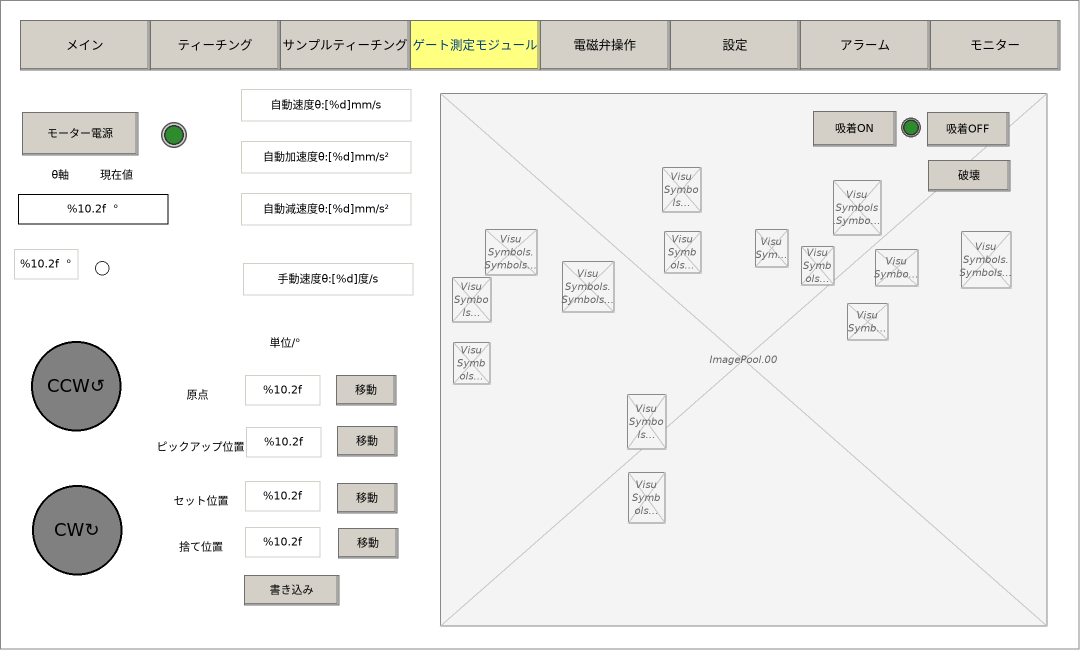
VISUALIZATION s_gm_teaching  // 1080x650
    Rectangle (0,0 1080x650)
    Label (35,160 51x30), "θ軸"
    Rectangle (18,194 150x30), "%10.2f °", text variable: gvl_axis.axisR.NcToPlc.ActPos
    Ellipse (31,341 90x90), "CCW↺", invisible if: gvl_axis.fbi_mc_powerR.Busy = FALSE
        OnMouseDown: execute { gvl_visu.flg_btn_rotaryRigt := true; }
        OnMouseUp: execute { gvl_visu.flg_btn_rotaryRigt := FALSE; }
    Ellipse (32,485 90x90), "CW↻", invisible if: gvl_axis.fbi_mc_powerR.Busy = FALSE
        OnMouseDown: execute { gvl_visu.flg_btn_rotaryLeft := TRUE; }
        OnMouseUp: execute { gvl_visu.flg_btn_rotaryLeft := FALSE; }
    Textfield (245,375 75x30), "%10.2f", text variable: gvl_visu.var_rotaryPos.origin
        OnMouseClick: write gvl_visu.var_rotaryPos.origin via VisuDialogs.Numpad
    Label (154,380 87x30), "原点"
    Textfield (246,427 75x30), "%10.2f", text variable: gvl_visu.var_rotaryPos.pickUp
        OnMouseClick: write gvl_visu.var_rotaryPos.pickUp via VisuDialogs.Numpad
    Label (159,432 83x30), "ピックアップ位置"
    Textfield (245,481 75x30), "%10.2f", text variable: gvl_visu.var_rotaryPos.set
        OnMouseClick: write gvl_visu.var_rotaryPos.set via VisuDialogs.Numpad
    Label (161,486 80x30), "セット位置"
    Lamp1 (159,120 30x30), variable: gvl_axis.fbi_mc_powerR.Busy, style: Lamp-Lamp1-Green
    Textfield (14,249 64x30), "%10.2f °", text variable: gvl_visu.var_gm_rotaryInch
        OnMouseClick: write gvl_visu.var_gm_rotaryInch via VisuDialogs.Numpad, format mm
    RadioButton (93,248 150x40), variable: gvl_visu.var_radio_rotaryJogMode
        Areas[0]: Text=インチ
        Areas[1]: Text=ジョグ
    Button (22,112 116x43), "モーター電源"
        toggle gvl_visu.flg_btn_gm_motorPower
    Button (244,575 95x30), "書き込み", colour toggle: gvl_visu.flg_btn_rotaryPos
        OnMouseClick: OpenDialog Dialog=d_gm_saveBtn, OpenModal=True, OpenCentered=True
    Button (336,375 60x30), "移動", invisible if: gvl_axis.fbi_mc_powerR.Busy = FALSE
        tap gvl_visu.flg_btn_gm_moveOrigin
    Button (337,426 60x30), "移動", invisible if: gvl_axis.fbi_mc_powerR.Busy = FALSE
        tap gvl_visu.flg_btn_gm_movePickUp
    Button (337,483 60x30), "移動", invisible if: gvl_axis.fbi_mc_powerR.Busy = FALSE
        tap gvl_visu.flg_btn_gm_moveSet
    Textfield (241,89 170x32), "自動速度θ:[%d]mm/s", text variable: gvl_visu.var_gm_autoRotaryVel
        OnMouseClick: write gvl_visu.var_gm_autoRotaryVel via VisuDialogs.Numpad
    Textfield (241,141 170x32), "自動加速度θ:[%d]mm/s²", text variable: gvl_visu.var_gm_autoRotaryAcc
        OnMouseClick: write gvl_visu.var_gm_autoRotaryAcc via VisuDialogs.Numpad
    Textfield (241,193 170x32), "自動減速度θ:[%d]mm/s²", text variable: gvl_visu.var_gm_autoRotaryDec
        OnMouseClick: write gvl_visu.var_gm_autoRotaryDec via VisuDialogs.Numpad
    Label (252,328 66x30), "単位/°"
    Label (91,160 51x30), "現在値"
    Textfield (243,263 170x32), "手動速度θ:[%d]度/s", text variable: gvl_visu.var_gm_manualRotaryVel
        OnMouseClick: write gvl_visu.var_gm_manualRotaryVel via VisuDialogs.Numpad
    Textfield (245,527 75x30), "%10.2f", text variable: gvl_visu.var_rotaryPos.remove
        OnMouseClick: write gvl_visu.var_rotaryPos.remove via VisuDialogs.Numpad
    Label (161,532 80x30), "捨て位置"
    Button (338,528 60x30), "移動", invisible if: gvl_axis.fbi_mc_powerR.Busy = FALSE
        tap gvl_visu.flg_btn_gm_moveRemove
    Image (440,93 607x533), image: ImagePool.00
    Image (562,261 52x51), angle 300, colour toggle: gvl_solv.ref_gm_rotary.in.in_flg_sensA, image: VisuSymbols.Symbols.ArrowQuarterLeftRight
        OnMouseDown: toggle gvl_visu.flg_btn_gm_svRotaryOrigin
    Image (485,229 52x46), angle 114, colour toggle: gvl_solv.ref_gm_rotary.in.in_flg_sensB, image: VisuSymbols.Symbols.ArrowQuarterRightLeft
        OnMouseDown: toggle gvl_visu.flg_btn_gm_svRotaryMoving
    Image (453,342 37x42), colour toggle: gvl_solv.ref_gm_pickUp.in.in_flg_sensA, image: VisuSymbols.Symbols.ArrowBoldDown
        OnMouseDown: toggle gvl_visu.flg_btn_gm_svPickUpOrigin
    Image (452,277 39x45), colour toggle: gvl_solv.ref_gm_pickUp.in.in_flg_sensB, image: VisuSymbols.Symbols.ArrowBoldUp
        OnMouseDown: toggle gvl_visu.flg_btn_gm_svPickUpMoving
    Image (801,246 33x39), angle 290, colour toggle: gvl_solv.ref_gm_chuck.in.in_flg_sensB, image: VisuSymbols.Symbols.ArrowBoldDown
        OnMouseDown: toggle gvl_visu.flg_btn_gm_svChuckClose
    Image (755,229 33x38), angle 290, colour toggle: gvl_solv.ref_gm_chuck.in.in_flg_sensA, image: VisuSymbols.Symbols.ArrowBoldUp
        OnMouseDown: toggle gvl_visu.flg_btn_gm_svChuckOpen
    Image (847,303 41x37), angle 343, colour toggle: gvl_solv.ref_gm_push.in.in_flg_sensB, image: VisuSymbols.Symbols.ArrowBoldLeftDown
        OnMouseDown: toggle gvl_visu.flg_btn_gm_svPushClose
    Image (875,249 43x37), angle 341, colour toggle: gvl_solv.ref_gm_push.in.in_flg_sensA, image: VisuSymbols.Symbols.ArrowBoldRightUp
        OnMouseDown: toggle gvl_visu.flg_btn_gm_svPushOpen
    Image (961,231 50x57), angle 290, colour toggle: gvl_solv.ref_gm_stamp.in.in_flg_sensB, image: VisuSymbols.Symbols.ArrowBoldDown
        OnMouseDown: toggle gvl_visu.flg_btn_gm_svStampMoving
    Image (833,180 48x55), angle 290, colour toggle: gvl_solv.ref_gm_stamp.in.in_flg_sensA, image: VisuSymbols.Symbols.ArrowBoldUp
        OnMouseDown: toggle gvl_visu.flg_btn_gm_svStampOrigin
    Image (627,394 39x55), colour toggle: gvl_elecylinder.ref_gm_axisTransport.input.in_flg_sensA, image: VisuSymbols.Symbols.ArrowBoldUp
        OnMouseDown: toggle gvl_visu.flg_btn_gm_eleTransportNegative
    Image (628,472 37x51), colour toggle: gvl_elecylinder.ref_gm_axisTransport.input.in_flg_sensB, image: VisuSymbols.Symbols.ArrowBoldDown
        OnMouseDown: toggle gvl_visu.flg_btn_gm_eleTransportPositive
    Image (662,167 39x45), colour toggle: gvl_elecylinder.ref_gm_axisPickUp.input.in_flg_sensA, image: VisuSymbols.Symbols.ArrowBoldUp
        OnMouseDown: toggle gvl_visu.flg_btn_gm_elePickUpNegative
    Image (664,231 37x42), colour toggle: gvl_elecylinder.ref_gm_axisPickUp.input.in_flg_sensB, image: VisuSymbols.Symbols.ArrowBoldDown
        OnMouseDown: toggle gvl_visu.flg_btn_gm_elePickUpPositive
    Button (813,111 83x35), "吸着ON"
        tap gvl_visu.flg_btn_gm_vacuumOn
    Button (928,160 82x31), "破壊"
        tap gvl_visu.flg_btn_gm_breakOn
    Button (927,112 82x34), "吸着OFF"
        tap gvl_visu.flg_btn_gm_vacuumOff
    Lamp1 (898,116 26x23), variable: gvl_solv.ref_gm_ejctor.input.in_flg_sensVac, style: Lamp-Lamp1-Green
    Button (20,20 130x50), "メイン"
        OnMouseClick: change screen: s_auto
    Button (150,20 130x50), "ティーチング"
        OnMouseClick: change screen: s_teaching1
    Button (670,20 130x50), "設定"
        OnMouseClick: change screen: s_setting
    Button (540,20 130x50), "電磁弁操作"
        OnMouseClick: change screen: s_manual
    Button (410,20 130x50), "ゲート測定モジュール"
        OnMouseClick: change screen: s_gm_teaching
    Button (800,20 130x50), "アラーム", colour toggle: gvl_io.flg_signalTowerRed
        OnMouseClick: change screen: s_alarm
    Button (280,20 130x50), "サンプルティーチング"
        OnMouseClick: change screen: s_sample
    Button (930,20 130x50), "モニター"
        OnMouseClick: change screen: s_monitor
END_VISUALIZATION

// ---- VISUs/Sheet/s_monitor.TcVIS
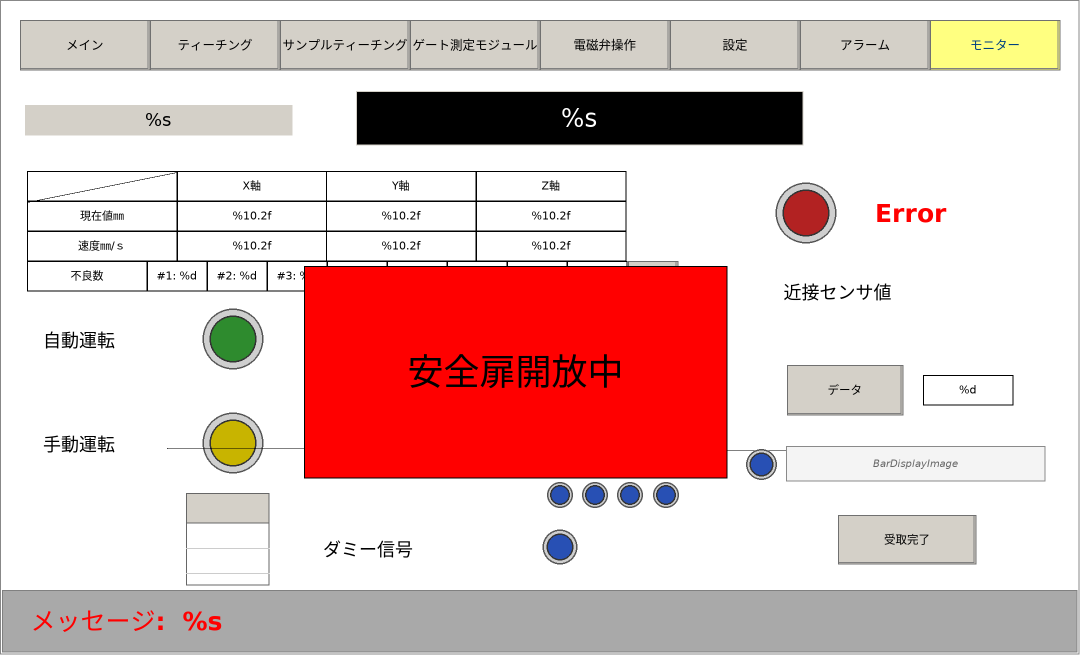
VISUALIZATION s_monitor  // 1080x655
    Rectangle (0,0 1080x655)
    Rectangle (177,201 150x30), "%10.2f", text variable: gvl_axis.axisX.NcToPlc.ActPos
    Rectangle (326,201 150x30), "%10.2f", text variable: gvl_axis.axisY.NcToPlc.ActPos
    Rectangle (476,201 150x30), "%10.2f", text variable: gvl_axis.axisZ.NcToPlc.ActPos
    Rectangle (177,171 150x30), "X軸"
    Rectangle (326,171 150x30), "Y軸"
    Rectangle (476,171 150x30), "Z軸"
    Rectangle (177,231 150x30), "%10.2f", text variable: gvl_axis.axisX.NcToPlc.ActVelo
    Rectangle (326,231 150x30), "%10.2f", text variable: gvl_axis.axisY.NcToPlc.ActVelo
    Rectangle (476,231 150x30), "%10.2f", text variable: gvl_axis.axisZ.NcToPlc.ActVelo
    Rectangle (27,171 150x30)
    Rectangle (27,201 150x30), "現在値㎜"
    Rectangle (27,231 150x30), "速度㎜/ｓ"
    Line (27,202) (177,172)
    Lamp1 (198,304 70x70), variable: gvl_param.var_currentMode = eP_programMode.auto, style: Lamp-Lamp1-Green
    Lamp1 (198,408 70x70), variable: gvl_param.var_currentMode = eP_programMode.manual, style: Lamp-Lamp1-Yellow
    Lamp1 (771,178 70x70), variable: gvl_param.var_currentMode = eP_programMode.error, invisible if: gvl_param.var_currentMode <> eP_programMode.error, style: Lamp-Lamp1-Red
    Label (839,194 144x38), "Error", invisible if: gvl_param.var_currentMode <> eP_programMode.error
    Line (167,448) (442,447)
    Line (560,451) (835,450)
    RoundedRectangle (25,105 267x30), "%s", text variable: gvl_visu.var_DT
    Rectangle (356,91 447x54), "%s", text variable: gvl_param.var_productInfo[gvl_param.var_currentProductID].name
    Button (628,261 50x30), "CLR"
        tap gvl_visu.flg_btn_clrDefectiveQty
    Rectangle (147,261 60x30), "#1: %d", text variable: gvl_auto.var_defectiveLens[1]
    Rectangle (267,261 60x30), "#3: %d", text variable: gvl_auto.var_defectiveLens[3]
    Rectangle (207,261 60x30), "#2: %d", text variable: gvl_auto.var_defectiveLens[2]
    Rectangle (327,261 60x30), "#4: %d", text variable: gvl_auto.var_defectiveLens[4]
    Rectangle (387,261 60x30), "#5: %d", text variable: gvl_auto.var_defectiveLens[5]
    Rectangle (447,261 60x30), "#6: %d", text variable: gvl_auto.var_defectiveLens[6]
    Rectangle (507,261 60x30), "#7: %d", text variable: gvl_auto.var_defectiveLens[7]
    Rectangle (567,261 60x30), "#8: %d", text variable: gvl_auto.var_defectiveLens[8]
    Rectangle (27,261 120x30), "不良数"
    Label (733,278 209x30), "近接センサ値"
    Rectangle (923,375 90x30), "%d", text variable: gvl_io.in_wire_gateLength
    Lamp1 (744,447 35x35), variable: gvl_auto.gateLengthIsPassed, style: Lamp-Lamp1-Blue
    Lamp1 (540,424 40x40), variable: gvl_IO.flg_gateLengthIsSuccessed, style: Lamp-Lamp1-Blue
    Lamp1 (540,370 40x40), variable: gvl_io.flg_lensSetDone, style: Lamp-Lamp1-Blue
    Lamp1 (545,480 30x30), variable: gvl_io.in_bitNumber3, style: Lamp-Lamp1-Blue
    Label (320,379 200x30), "レンズセット完了信号"
    Label (320,430 200x30), "ゲート測定OK信号"
    Rectangle (40,326 140x30), "自動運転", text variable: gvl_auto.cavNo
    Label (320,328 200x30), "レンズ要求信号"
    Lamp1 (540,323 40x40), variable: gvl_io.flg_requestLens, style: Lamp-Lamp1-Red
    Lamp1 (540,527 40x40), variable: gvl_io.flg_dummySiganl, style: Lamp-Lamp1-Blue
    Lamp1 (580,480 30x30), variable: gvl_io.flg_bitNumber2, style: Lamp-Lamp1-Blue
    Lamp1 (615,480 30x30), variable: gvl_io.flg_bitNumber1, style: Lamp-Lamp1-Blue
    Lamp1 (651,480 30x30), variable: gvl_io.flg_bitNumber0, style: Lamp-Lamp1-Blue
    Label (529,457 165x30), "4 3 2 1"
    Label (320,535 200x30), "ダミー信号"
    Table (186,493 83x92), data array: gvl_auto.pocketNo
        p3854506369: gvl_auto.pocketNo[INDEX]
    Button (20,20 130x50), "メイン"
        OnMouseClick: change screen: s_auto
    Button (150,20 130x50), "ティーチング"
        OnMouseClick: change screen: s_teaching1
    Button (670,20 130x50), "設定"
        OnMouseClick: change screen: s_setting
    Button (540,20 130x50), "電磁弁操作"
        OnMouseClick: change screen: s_manual
    Button (410,20 130x50), "ゲート測定モジュール"
        OnMouseClick: change screen: s_gm_teaching
    Button (800,20 130x50), "アラーム", colour toggle: gvl_io.flg_signalTowerRed
        OnMouseClick: change screen: s_alarm
    Button (280,20 130x50), "サンプルティーチング"
        OnMouseClick: change screen: s_sample
    BarDisplayImage (786,446 259x35), value: gvl_visu.var_curenntGateData, style: BarDisplayImage-Gray, scale format: %.1f, scale 0..3
    Button (787,365 116x50), "データ"
        OnMouseClick: change screen: s_gateLengthData
    Rectangle (304,266 423x212), "安全扉開放中", text variable: gvl_io.flg_frontSaftyDoor or gvl_param.var_currentMode <> eP_programMode.auto, invisible if: gvl_io.flg_frontSaftyDoor or gvl_param.var_currentMode <> eP_programMode.auto
    Button (930,20 130x50), "モニター"
        OnMouseClick: change screen: s_monitor
    Rectangle (40,430 140x30), "手動運転", text variable: gvl_auto.cavNo
    Button (838,515 138x49), "受取完了", invisible if: gvl_debug.flg_debug_run = FALSE OR gvl_io.flg_requestLens = FALSE
        tap gvl_visu.flg_btn_lensSetDone
    Rectangle (2,590 1075x62), "メッセージ: %s", text variable: gvl_visu.var_msg
END_VISUALIZATION

// ---- VISUs/Sheet/s_sample.TcVIS
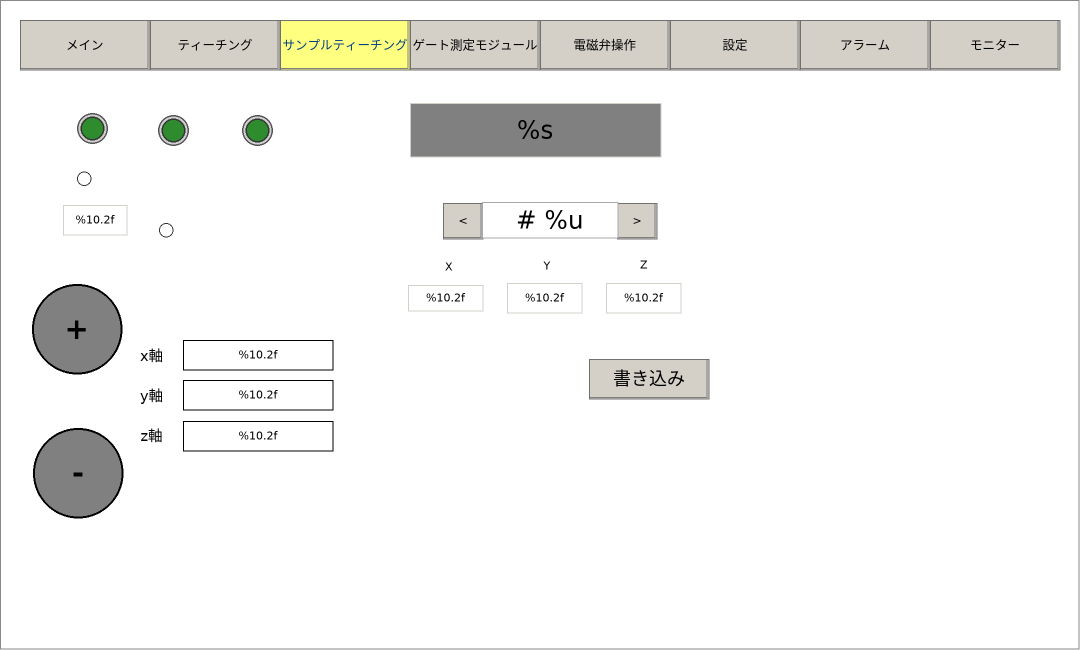
VISUALIZATION s_sample  // 1080x650
    Rectangle (0,0 1080x650)
    Lamp1 (240,113 35x35), variable: gvl_axis.fbi_mc_powerZ.Busy, style: Lamp-Lamp1-Green
    Lamp1 (156,113 35x35), variable: gvl_axis.fbi_mc_powerY.Busy, style: Lamp-Lamp1-Green
    Lamp1 (75,111 35x35), variable: gvl_axis.fbi_mc_powerX.Busy, style: Lamp-Lamp1-Green
    Textfield (63,205 64x30), "%10.2f", text variable: gvl_visu.var_in_inch
        OnMouseClick: write gvl_visu.var_in_inch via VisuDialogs.Numpad, format mm
    Label (126,341 51x30), "x軸"
    Label (126,381 51x30), "y軸"
    Label (126,421 51x30), "z軸"
    Rectangle (183,340 150x30), "%10.2f", text variable: gvl_axis.AxisX.NcToPlc.ActPos
    Rectangle (183,380 150x30), "%10.2f", text variable: gvl_axis.AxisY.NcToPlc.ActPos
    Rectangle (183,421 150x30), "%10.2f", text variable: gvl_axis.AxisZ.NcToPlc.ActPos
    RadioButton (75,159 249x39), variable: gvl_visu.var_jofAxis
    RadioButton (157,210 169x40), variable: gvl_visu.var_radio_jogMode
        Areas[0]: Text=インチ
        Areas[1]: Text=ジョグ
    Ellipse (32,284 90x90), "+", invisible if: gvl_axis.flg_motorReady = FALSE
        OnMouseDown: execute { gvl_visu.flg_btn_moveDirct := eP_direction.positive; }
        OnMouseUp: execute { gvl_visu.flg_btn_moveDirct := eP_direction.keep; }
    Ellipse (33,428 90x90), "-", invisible if: gvl_axis.flg_motorReady = FALSE
        OnMouseDown: execute { gvl_visu.flg_btn_moveDirct := eP_direction.negative; }
        OnMouseUp: execute { gvl_visu.flg_btn_moveDirct := eP_direction.keep; }
    Textfield (408,285 75x26), "%10.2f", text variable: gvl_visu.var_in_samplePos.x
        OnMouseClick: write gvl_visu.var_in_samplePos.x via VisuDialogs.Numpad
    Textfield (507,283 75x30), "%10.2f", text variable: gvl_visu.var_in_samplePos.y
        OnMouseClick: write gvl_visu.var_in_samplePos.y via VisuDialogs.Numpad
    Textfield (606,283 75x30), "%10.2f", text variable: gvl_visu.var_in_samplePos.z
        OnMouseClick: write gvl_visu.var_in_samplePos.z via VisuDialogs.Numpad
    Label (424,252 50x30), "X"
    Label (522,251 50x30), "Y"
    Label (619,250 50x30), "Z"
    Rectangle (410,103 251x54), "%s", text variable: gvl_param.var_productInfo[gvl_param.var_currentProductID].name
    Button (589,359 120x40), "書き込み"
        OnMouseClick: OpenDialog Dialog=d_saveSample, OpenModal=True, OpenCentered=True
    Button (20,20 130x50), "メイン"
        OnMouseClick: change screen: s_auto
    Button (150,20 130x50), "ティーチング"
        OnMouseClick: change screen: s_teaching1
    Button (670,20 130x50), "設定"
        OnMouseClick: change screen: s_setting
    Button (540,20 130x50), "電磁弁操作"
        OnMouseClick: change screen: s_manual
    Button (410,20 130x50), "ゲート測定モジュール"
        OnMouseClick: change screen: s_gm_teaching
    Button (800,20 130x50), "アラーム", colour toggle: gvl_io.flg_signalTowerRed
        OnMouseClick: change screen: s_alarm
    Button (280,20 130x50), "サンプルティーチング"
        OnMouseClick: change screen: s_sample
    Button (617,203 40x36), ">"
        OnMouseClick: execute {
            IF gvl_visu.var_in_sampleCavNo < 8 THEN
            	gvl_visu.var_in_sampleCavNo := gvl_visu.var_in_sampleCavNo + 1;
            END_IF
        }
    Button (443,203 40x36), "<"
        OnMouseClick: execute {
            IF gvl_visu.var_in_sampleCavNo > 1 THEN
            	gvl_visu.var_in_sampleCavNo := gvl_visu.var_in_sampleCavNo - 1;
            END_IF
        }
    Rectangle (482,202 136x36), "# %u", text variable: gvl_visu.var_in_sampleCavNo
    Button (930,20 130x50), "モニター"
        OnMouseClick: change screen: s_monitor
END_VISUALIZATION

// ---- VISUs/Sheet/s_setting.TcVIS
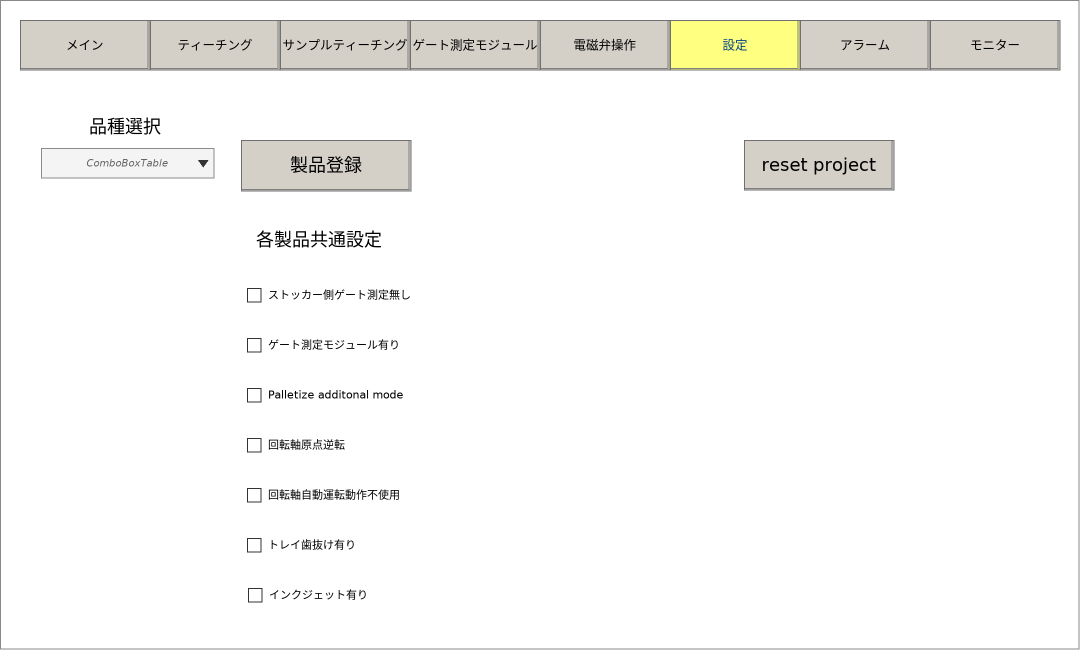
VISUALIZATION s_setting  // 1080x650
    Rectangle (0,0 1080x650)
    Label (50,112 150x30), "品種選択"
    ComboBoxTable (41,148 173x30), variable: gvl_param.var_currentProductID, data array: gvl_visu.var_in_currentProduct
        p3854506369: gvl_visu.var_in_currentProduct[INDEX]
    Checkbox (245,280 400x30), "ストッカー側ゲート測定無し", variable: gvl_visu.flg_btn_gateMeasurementIsNone
    Checkbox (245,330 400x30), "ゲート測定モジュール有り", variable: gvl_visu.flg_btn_usingMeasurementSystem
    Button (241,140 170x51), "製品登録"
        OnMouseClick: change screen: s_addNewProduct
    Checkbox (245,380 400x30), "Palletize additonal mode", variable: gvl_visu.var_dev_palletizingMode
    Button (20,20 130x50), "メイン"
        OnMouseClick: change screen: s_auto
    Button (150,20 130x50), "ティーチング"
        OnMouseClick: change screen: s_teaching1
    Button (670,20 130x50), "設定"
        OnMouseClick: change screen: s_setting
    Button (540,20 130x50), "電磁弁操作"
        OnMouseClick: change screen: s_manual
    Button (410,20 130x50), "ゲート測定モジュール"
        OnMouseClick: change screen: s_gm_teaching
    Button (800,20 130x50), "アラーム", colour toggle: gvl_io.flg_signalTowerRed
        OnMouseClick: change screen: s_alarm
    Button (280,20 130x50), "サンプルティーチング"
        OnMouseClick: change screen: s_sample
    Button (744,140 150x50), "reset project"
        OnMouseClick: OpenDialog Dialog=d_resetProject, OpenModal=True, OpenCentered=True
    Checkbox (245,430 400x30), "回転軸原点逆転", variable: gvl_visu.flg_btn_rotaryReversal
    Checkbox (245,480 400x30), "回転軸自動運転動作不使用", variable: gvl_visu.flg_btn_RotaryIsNotUse
    Checkbox (245,530 400x30), "トレイ歯抜け有り", variable: gvl_visu.flg_missingParts
    Checkbox (246,580 400x30), "インクジェット有り", variable: gvl_visu.flg_usingTimeStamp
    Button (930,20 130x50), "モニター"
        OnMouseClick: change screen: s_monitor
    Label (253,213 189x54), "各製品共通設定"
END_VISUALIZATION

// ---- VISUs/Sheet/s_teaching1.TcVIS
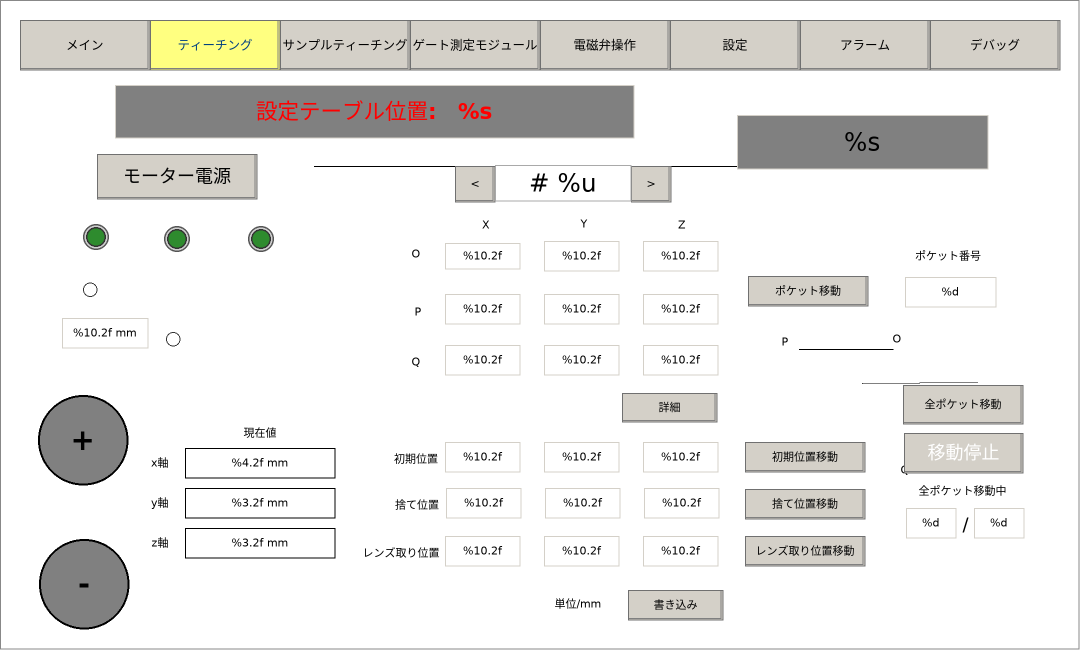
VISUALIZATION s_teaching1  // 1080x650
    Rectangle (0,0 1080x650)
    Lamp1 (246,224 30x30), variable: gvl_axis.fbi_mc_powerZ.Busy, style: Lamp-Lamp1-Green
    Lamp1 (162,224 30x30), variable: gvl_axis.fbi_mc_powerY.Busy, style: Lamp-Lamp1-Green
    Lamp1 (81,222 30x30), variable: gvl_axis.fbi_mc_powerX.Busy, style: Lamp-Lamp1-Green
    Textfield (445,243 75x26), "%10.2f", text variable: gvl_visu.var_in_palletizePos.Pos[1].x
        OnMouseClick: write gvl_visu.var_in_palletizePos.Pos[1].x via VisuDialogs.Numpad
    Textfield (445,294 75x30), "%10.2f", text variable: gvl_visu.var_in_palletizePos.Pos[2].x
        OnMouseClick: write gvl_visu.var_in_palletizePos.Pos[2].x via VisuDialogs.Numpad
    Textfield (445,345 75x30), "%10.2f", text variable: gvl_visu.var_in_palletizePos.Pos[3].x
        OnMouseClick: write gvl_visu.var_in_palletizePos.Pos[3].x via VisuDialogs.Numpad
    Label (391,347 50x30), "Q"
    Label (391,239 50x30), "O"
    Label (393,297 50x30), "P"
    Group (760,324 120x92)
        Line (39,25) (133,25)
        Line (102,59) (217,58)
        Label (112,0 50x30), "O"
        Label (0,3 50x30), "P"
        Label (120,131 50x30), "Q"
    Button (628,590 95x30), "書き込み"
        OnMouseClick: OpenDialog Dialog=d_saveBtn, OpenModal=True, OpenCentered=True
    Line (314,166) (799,166)
    Label (906,241 84x30), "ポケット番号", invisible if: gvl_visu.flg_All_PosPorket_Move
    Button (748,276 120x30), "ポケット移動", invisible if: gvl_axis.flg_motorReady = FALSE OR gvl_visu.flg_All_PosPorket_Move
        tap gvl_visu.flg_btn_PosPocket
    Textfield (62,318 86x30), "%10.2f mm", text variable: gvl_visu.var_in_inch
        OnMouseClick: write gvl_visu.var_in_inch via VisuDialogs.Numpad
    Textfield (544,241 75x30), "%10.2f", text variable: gvl_visu.var_in_palletizePos.Pos[1].y
        OnMouseClick: write gvl_visu.var_in_palletizePos.Pos[1].y via VisuDialogs.Numpad
    Textfield (643,241 75x30), "%10.2f", text variable: gvl_visu.var_in_palletizePos.Pos[1].z
        OnMouseClick: write gvl_visu.var_in_palletizePos.Pos[1].z via VisuDialogs.Numpad
    Textfield (544,294 75x30), "%10.2f", text variable: gvl_visu.var_in_palletizePos.Pos[2].y
        OnMouseClick: write gvl_visu.var_in_palletizePos.Pos[2].y via VisuDialogs.Numpad
    Textfield (643,294 75x30), "%10.2f", text variable: gvl_visu.var_in_palletizePos.Pos[2].z
        OnMouseClick: write gvl_visu.var_in_palletizePos.Pos[2].z via VisuDialogs.Numpad
    Textfield (544,345 75x30), "%10.2f", text variable: gvl_visu.var_in_palletizePos.Pos[3].y
        OnMouseClick: write gvl_visu.var_in_palletizePos.Pos[3].y via VisuDialogs.Numpad
    Textfield (643,345 75x30), "%10.2f", text variable: gvl_visu.var_in_palletizePos.Pos[3].z
        OnMouseClick: write gvl_visu.var_in_palletizePos.Pos[3].z via VisuDialogs.Numpad
    Label (461,210 50x30), "X"
    Label (559,209 50x30), "Y"
    Label (657,210 50x30), "Z"
    Textfield (445,442 75x30), "%10.2f", text variable: gvl_visu.var_in_initialPos.x
        OnMouseClick: write gvl_visu.var_in_initialPos.x via VisuDialogs.Numpad
    Label (391,444 50x30), "初期位置"
    Textfield (544,442 75x30), "%10.2f", text variable: gvl_visu.var_in_initialPos.y
        OnMouseClick: write gvl_visu.var_in_initialPos.y via VisuDialogs.Numpad
    Textfield (643,442 75x30), "%10.2f", text variable: gvl_visu.var_in_initialPos.z
        OnMouseClick: write gvl_visu.var_in_initialPos.z via VisuDialogs.Numpad
    Textfield (446,488 75x30), "%10.2f", text variable: gvl_visu.var_in_removePos.x
        OnMouseClick: write gvl_visu.var_in_removePos.x via VisuDialogs.Numpad
    Label (392,490 50x30), "捨て位置"
    Textfield (545,488 75x30), "%10.2f", text variable: gvl_visu.var_in_removePos.y
        OnMouseClick: write gvl_visu.var_in_removePos.y via VisuDialogs.Numpad
    Textfield (644,488 75x30), "%10.2f", text variable: gvl_visu.var_in_removePos.z
        OnMouseClick: write gvl_visu.var_in_removePos.z via VisuDialogs.Numpad
    Textfield (445,536 75x30), "%10.2f", text variable: gvl_visu.var_in_pickUpPos.x
        OnMouseClick: write gvl_visu.var_in_pickUpPos.x via VisuDialogs.Numpad
    Label (361,538 80x30), "レンズ取り位置"
    Textfield (544,536 75x30), "%10.2f", text variable: gvl_visu.var_in_pickUpPos.y
        OnMouseClick: write gvl_visu.var_in_pickUpPos.y via VisuDialogs.Numpad
    Textfield (643,536 75x30), "%10.2f", text variable: gvl_visu.var_in_pickUpPos.z
        OnMouseClick: write gvl_visu.var_in_pickUpPos.z via VisuDialogs.Numpad
    Button (745,442 120x30), "初期位置移動", invisible if: gvl_axis.flg_motorReady = FALSE
        tap gvl_visu.flg_btn_PosInit
    Button (745,489 120x30), "捨て位置移動", invisible if: gvl_axis.flg_motorReady = FALSE
        tap gvl_visu.flg_btn_PosRemove
    Button (745,536 120x30), "レンズ取り位置移動", invisible if: gvl_axis.flg_motorReady = FALSE
        tap gvl_visu.flg_btn_PosPickUP
    Label (135,448 50x30), "x軸"
    Label (135,488 50x30), "y軸"
    Label (135,528 50x30), "z軸"
    Rectangle (185,448 150x30), "%4.2f mm", text variable: gvl_axis.AxisX.NcToPlc.ActPos
    Rectangle (185,488 150x30), "%3.2f mm", text variable: gvl_axis.AxisY.NcToPlc.ActPos
    Rectangle (185,528 150x30), "%3.2f mm", text variable: gvl_axis.AxisZ.NcToPlc.ActPos
    RadioButton (81,270 249x39), variable: gvl_visu.var_jofAxis
    RadioButton (164,319 169x40), variable: gvl_visu.var_radio_jogMode
        Areas[0]: Text=インチ
        Areas[1]: Text=ジョグ
    Rectangle (737,115 251x54), "%s", text variable: gvl_param.var_productInfo[gvl_param.var_currentProductID].name
    Rectangle (115,85 519x53), "設定テーブル位置: %s", text variable: gvl_visu.var_currentTableMsg
    Ellipse (38,395 90x90), "+", invisible if: gvl_axis.flg_motorReady = FALSE
        OnMouseDown: execute { gvl_visu.flg_btn_moveDirct := eP_direction.positive; }
        OnMouseUp: execute { gvl_visu.flg_btn_moveDirct := eP_direction.keep; }
    Ellipse (39,539 90x90), "-", invisible if: gvl_axis.flg_motorReady = FALSE
        OnMouseDown: execute { gvl_visu.flg_btn_moveDirct := eP_direction.negative; }
        OnMouseUp: execute { gvl_visu.flg_btn_moveDirct := eP_direction.keep; }
    Textfield (905,277 91x30), "%d", text variable: gvl_visu.var_in_pocketNo, invisible if: gvl_visu.flg_All_PosPorket_Move
        OnMouseClick: write gvl_visu.var_in_pocketNo via VisuDialogs.Numpad
    Button (97,154 160x45), "モーター電源"
        toggle gvl_visu.flg_powerOn
    Button (622,393 95x29), "詳細"
        OnMouseClick: OpenDialog Dialog=d_teahingDetail, OpenModal=True, OpenCentered=True
    Button (20,20 130x50), "メイン"
        OnMouseClick: change screen: s_auto
    Button (150,20 130x50), "ティーチング"
        OnMouseClick: change screen: s_teaching1
    Button (670,20 130x50), "設定"
        OnMouseClick: change screen: s_setting
    Button (540,20 130x50), "電磁弁操作"
        OnMouseClick: change screen: s_manual
    Button (410,20 130x50), "ゲート測定モジュール"
        OnMouseClick: change screen: s_gm_teaching
    Button (800,20 130x50), "アラーム", colour toggle: gvl_io.flg_signalTowerRed
        OnMouseClick: change screen: s_alarm
    Button (280,20 130x50), "サンプルティーチング"
        OnMouseClick: change screen: s_sample
    Button (631,166 40x36), ">"
        OnMouseClick: execute {
            IF gvl_visu.var_in_cavNo < 8 THEN
            	gvl_visu.var_in_cavNo := gvl_visu.var_in_cavNo + 1;
            END_IF
        }
    Button (455,166 40x36), "<"
        OnMouseClick: execute {
            IF gvl_visu.var_in_cavNo > 1 THEN
            	gvl_visu.var_in_cavNo := gvl_visu.var_in_cavNo - 1;
            END_IF
        }
    Rectangle (495,165 136x36), "# %u", text variable: gvl_visu.var_in_cavNo
    Label (545,589 66x30), "単位/mm"
    Label (235,418 50x30), "現在値"
    Button (930,20 130x50), "デバッグ", colour toggle: gvl_io.flg_signalTowerRed
        OnMouseClick: change screen: s_debug
    Button (903,385 120x39), "全ポケット移動", invisible if: gvl_axis.flg_motorReady = FALSE OR gvl_visu.flg_All_PosPorket_Move
        tap gvl_visu.flg_btn_All_PosPocket
    Button (904,433 119x40), "移動停止", text variable: gvl_text.var_stopping, colour toggle: gvl_visu.flg_btn_autoModeStop, invisible if: NOT gvl_visu.flg_All_PosPorket_Move
        tap gvl_visu.flg_btn_autoModeStop
    Label (953,509 25x31), "/", invisible if: NOT gvl_visu.flg_All_PosPorket_Move
    Textfield (906,508 50x30), "%d", text variable: gvl_visu.var_in_pocketNo, invisible if: NOT gvl_visu.flg_All_PosPorket_Move
        OnMouseClick: write the text variable via VisuDialogs.Numpad
    Textfield (974,508 50x30), "%d", text variable: gvl_param.var_productInfo[gvl_param.var_currentProductID].pocketSumQty, invisible if: NOT gvl_visu.flg_All_PosPorket_Move
        OnMouseClick: write the text variable via VisuDialogs.Numpad
    Label (908,476 109x30), "全ポケット移動中", invisible if: NOT gvl_visu.flg_All_PosPorket_Move
END_VISUALIZATION
